TYPE Udt_CM_Sensor2State :
STRUCT
	sensor_Input : BOOL;
	
	sensor_Output : BOOL; 
END_STRUCT
END_TYPE

(* stored: Version 1.1.0.1, ProductVersion 3.1.4024.13
   DUT Udt_CM_Sensor2State: Id {bb0fd379-6075-4547-b4b5-3304d175e36a} *)
